// Mitsubishi GX Works2 project: BacNinhTapFX3S   PLC: FX3S

// global labels: Global1
VAR_GLOBAL
  VR1 AT D8030 : INT;
  VR2 AT D8031 : INT;
  XXLimitN AT M8344 : BOOL;
  XXLimitP AT M8343 : BOOL;
  XXBusy AT M8340 : BOOL;
  XXInterruptInverse AT M8347 : BOOL;
  XXPos AT D8340 : DINT;
  XXAccelTime AT D8348 : INT;
  XXDecelTime AT D8349 : INT;
  XXPosView AT D0 : DINT;
  XXTarPos AT D2 : DINT;
  XXFeed AT D4 : DINT;
  XXTarR AT M0 : BOOL;
  XXTarRSkip AT D6 : INT;
  XXOn AT M1 : BOOL;
  XXRun AT M2 : BOOL;
  XXDirection AT M3 : BOOL;
  XXMinI AT X000 : BOOL;
  XXMaxI AT X001 : BOOL;
  XXReadyI AT X002 : BOOL;
  XXPulseO AT Y000 : BOOL;
  XXDirectionO AT Y004 : BOOL;
  XXOnO AT Y002 : BOOL;
  Run AT M4 : BOOL;
  RunI AT X003 : BOOL;
  RunStop AT M5 : BOOL;
  RunStopI AT X004 : BOOL;
  RunState AT D7 : INT;
  RunStateNext AT M6 : BOOL;
  AxisState AT D8 : INT;
  AxisStateNext AT M7 : BOOL;
  FoilState AT D9 : INT;
  FoilStateNext AT M8 : BOOL;
  FoilTopN AT M9 : BOOL;
  FoilTopNI AT X005 : BOOL;
  FoilTopP AT M10 : BOOL;
  FoilTopPI AT X006 : BOOL;
  FoilTopTimer AT TC0 : BOOL;
  FoilTopTimerDelay AT D10 : INT;
  FoilTop AT M11 : BOOL;
  FoilTopO AT Y005 : BOOL;
  FoilBotN AT M12 : BOOL;
  FoilBotNI AT X007 : BOOL;
  FoilBotP AT M13 : BOOL;
  FoilBotPI AT X010 : BOOL;
  FoilBotTimer AT TC1 : BOOL;
  FoilBotTimerDelay AT D11 : INT;
  FoilBot AT M14 : BOOL;
  FoilBotO AT Y006 : BOOL;
  WorkFeed AT D12 : DINT;
END_VAR

// task Task_01 (event TRUE, interval 0, priority 31): POU_01

PROGRAM POU_01
VAR
  fTmp : BOOL;
END_VAR
RST(M8002, XXOn);
MOV(M8002, 200, XXAccelTime);
MOV(M8002, 200, XXDecelTime);
SET(M8002, FoilTop);
SET(M8002, FoilBot);
(*1000 pulse = 1 mm, 1 round = 1.75mm, -> servo ppr = 1750*)
DMOV(M8002, (1750 * 2000) / 60, WorkFeed);
(*|||||||||||||||*)
(*|||||||||||||||*)
SET(Run AND RunState = 0, fTmp);
RST(fTmp, Run);
SET(fTmp, XXOn);
MOV(fTmp, 1, RunState);
RST(fTmp, fTmp);
SET(RunStop, fTmp);
RST(fTmp, Run);
RST(fTmp, RunStop);
ZRST(fTmp, RunState, FoilState);
RST(fTmp, XXRun);
RST(fTmp, XXOn);
SET(fTmp, FoilTop);
SET(fTmp, FoilBot);
RST(fTmp, fTmp);
(*|||||||||||||||*)
(*|||||||||||||||*)
INC(RunStateNext, RunState);
INC(AxisStateNext, AxisState);
INC(FoilStateNext, FoilState);
ZRST(M8000, RunStateNext, FoilStateNext);
DECO(M8000, RunState, 6, M100);
DECO(M8000, AxisState, 6, M200); DECO(M8000, AxisState, 6, M1200); ZRST(NOT XXTarR OR NOT XXReadyI, M1200, M1263);
DECO(M8000, FoilState, 6, M300);
(*|||||||||||||||*)

(*|||||||||||||||*)
(*origin*)
MOV(M101, 1, AxisState);
MOV(M101, 1, FoilState);
SET(M101, RunStateNext);
(*ready done*)
SET(M102 AND M1220 AND M320, RunStateNext);
(*tap*)
MOV(M103, 11, AxisState);
SET(M103, RunStateNext);
(*tap done, drop*)
MOV(M104 AND M1220, 11, FoilState);
SET(M104 AND M1220, RunStateNext);
(*drop done, back to ready*)
MOV(M105, 2, RunState);
(*|||||||||||||||*)

(*|||||||||||||||*)
(*/////get origin*)
(*at min, jump to move down*)
SET(M1201 AND XXMinI, fTmp);
MOV(fTmp, 3, AxisState); RST(fTmp, fTmp);
(*not at min, move up*)
SET(M1201 AND NOT XXMinI, fTmp);
RST(fTmp, XXPos);
DMOV(fTmp, -50_000, XXTarPos);
DMOV(fTmp, 5_000, XXFeed);
SET(fTmp, XXRun);
SET(fTmp, AxisStateNext); RST(fTmp, fTmp);
(*move up hit limit, reset*)
SET(M202 AND NOT XXBusy, fTmp);
RST(fTmp, XXRun);
RST(fTmp, XXPos);
SET(fTmp, AxisStateNext); RST(fTmp, fTmp);
(*move down*)
SET(M1203, fTmp);
DMOV(fTmp, 5_000, XXTarPos);
DMOV(fTmp, 1_000, XXFeed);
SET(fTmp, XXRun);
SET(fTmp, AxisStateNext); RST(fTmp, fTmp);
(*move down out min, stop*)
SET(M204 AND NOT XXMinI, fTmp);
RST(fTmp, XXRun);
SET(fTmp, AxisStateNext); RST(fTmp, fTmp);
(*stop done, move down 1mm*)
SET(M1205, fTmp);
DMOV(fTmp, XXPos + 1000, XXTarPos);
DMOV(fTmp, 1000, XXFeed);
SET(fTmp, XXRun);
SET(fTmp, AxisStateNext); RST(fTmp, fTmp);
(*move down 1mm done, ready*)
SET(M1206, fTmp);
RST(fTmp, XXPos);
MOV(fTmp, 20, AxisState); RST(fTmp, fTmp);
(*/////main sequence*)
(*wait run hit, move down*)
SET(M1211 AND Run, fTmp);
DMOV(fTmp, 35_000, XXTarPos);
DMOV(fTmp, WorkFeed, XXFeed);
SET(fTmp, XXRun);
SET(fTmp, AxisStateNext); RST(fTmp, fTmp);
(*target reach or touch max, reset*)
SET(M1212 OR (M212 AND NOT XXBusy), fTmp);
RST(fTmp, XXRun);
SET(fTmp, AxisStateNext); RST(fTmp, fTmp);
(*move down slow done, move up*)
SET(M1213, fTmp);
DMOV(fTmp, 0, XXTarPos);
DMOV(fTmp, WorkFeed, XXFeed);
SET(fTmp, XXRun);
SET(fTmp, AxisStateNext); RST(fTmp, fTmp);
(*move up done, return wait tap hit*)
SET(M1214, fTmp);
MOV(fTmp, 20, AxisState); RST(fTmp, fTmp);
(*|||||||||||||||*)

(*|||||||||||||||*)
MOV(M8000, 1 + (VR1 / 16), FoilTopTimerDelay);
MOV(M8000, 1 + (VR2 / 16), FoilBotTimerDelay);
(*get origin*)
SET(M301, FoilTop);
SET(M301, FoilBot);
SET(M301 AND FoilTopP AND FoilBotP, FoilStateNext);
(*get origin done*)
MOV(M302, 20, FoilState);
(*/////main sequence*)
(*bot back, done, next*)
RST(M311, FoilBot);
SET(M311 AND FoilBotN, FoilStateNext);
(*wait drop, bot forward, done, next*)
OUT_T(M312, FoilBotTimer, FoilBotTimerDelay);
SET(FoilBotTimer, FoilBot);
SET(FoilBotTimer AND FoilBotP, FoilStateNext);
(*top back, done, next*)
RST(M313, FoilTop);
SET(M313 AND FoilTopN, FoilStateNext);
(*wait drop, top forward, done, next*)
OUT_T(M314, FoilTopTimer, FoilTopTimerDelay);
SET(FoilTopTimer, FoilTop);
SET(FoilTopTimer AND FoilTopP, FoilStateNext);
(*end*)
MOV(M315, 20, FoilState);
(*|||||||||||||||*)

(*|||||||||||||||*)
(*XX*)
RST(XXRun AND XXTarPos = XXPos, XXRun);
DDRVA(XXRun, XXTarPos, XXFeed, XXPulseO, XXDirection);
RST(M8029, XXRun);
OUT(XXDirection, XXDirectionO);
INC(NOT XXRun AND NOT XXBusy AND XXTarRSkip < 5, XXTarRSkip);
RST(XXRun, XXTarRSkip);
OUT(XXTarRSkip >= 5, XXTarR);
(**)
OUT(XXMinI, XXLimitN);
OUT(XXMaxI, XXLimitP);
(*|||||||||||||||*)

(*|||||||||||||||*)
PLS(RunI, Run); SET(Run, Run);
PLS(RunStopI, RunStop); SET(RunStop, RunStop);
SET(FoilTopNI, FoilTopN); RST(FoilTopNI, FoilTopP);
SET(FoilTopPI, FoilTopP); RST(FoilTopPI, FoilTopN);
SET(FoilBotNI, FoilBotN); RST(FoilBotNI, FoilBotP);
SET(FoilBotPI, FoilBotP); RST(FoilBotPI, FoilBotN);
(*|||||||||||||||*)
OUT(XXOn, XXOnO);
OUT(NOT FoilTop, FoilTopO);
OUT(NOT FoilBot, FoilBotO);
(*|||||||||||||||*)
END_PROGRAM
